(* IEC 61131-3 sources: windowtracking/test, 11 files *)

(* ---- ClearWindowTest.st ---- *)
USING AxUnit.Assert;
USING Simatic.Ax.WindowTracking.EventHandler;
USING Simatic.Ax.WindowTracking.Trigger;

NAMESPACE Simatic.Ax.WindowTracking.EventHandler
    {TestFixture}
    CLASS ClearWindowTest
        VAR PROTECTED
            tws : TransportWindowList;
            enc : EncoderMock;
            v1 : VirtualTrigger := (Position := 100, Id := UINT#1);
            v2 : VirtualTrigger := (Position := 200, Id := UINT#2);
            te1 : TriggerEventMock;
            te2 : TerminateWindowEvent;
            tl : TriggerList;
        END_VAR

        METHOD PROTECTED Setup
            tws.Encoder := enc;
            v1.EventHandler := te1;
            v2.EventHandler := te2;
            te2.WindowList := tws;
            tl.Add(v1);
            tl.Add(v2);
            tws.TriggerPointList := tl;
        END_METHOD

        {Test}
        METHOD PUBLIC Test_Clear_window
            THIS.Setup();
            tws.Create();
            enc.EncoderValue := 0;
            tws.Evaluate();
            Equal(expected := UINT#1, actual := tws.Count());

            enc.EncoderValue := 100;
            tws.Create();
            tws.Evaluate();
            Equal(expected := UINT#2, actual := tws.Count());

            // Remove Window at Position 200
            enc.EncoderValue := 200;
            tws.Evaluate();
            Equal(expected := UINT#1, actual := tws.Count());

        END_METHOD
    END_CLASS
END_NAMESPACE

(* ---- ItemTest.st ---- *)
USING AxUnit.Assert;
USING Simatic.Ax.WindowTracking.Trigger;

NAMESPACE Simatic.Ax.WindowTracking.Items
    {TestFixture}
    CLASS ItemTest
        VAR PROTECTED
            i : ItemOneDestination;
            vt : VirtualTrigger;
            ivt : IVirtualTrigger;
        END_VAR

        {Test}
        METHOD PUBLIC Test_Count_with_no_deststination_expect_0
            Equal(expected := i.DestinationCount(), actual := 0);
        END_METHOD

        {Test}
        METHOD PUBLIC Test_Count_with_1_deststination_expect_1
            i.Destination1 := vt;
            Equal(expected := i.DestinationCount(), actual := 1);
        END_METHOD

        {Test}
        METHOD PUBLIC Test_GetItem_with_no_deststination_expect_NULL
            Equal(expected := TRUE, actual := i.GetDestination() = NULL);
        END_METHOD

        {Test}
        METHOD PUBLIC Test_GetItem_with_1_deststination_expect_desztiation
            i.Destination1 := vt;
            ivt := vt;
            Equal(expected := TRUE, actual := i.GetDestination() = ivt);
        END_METHOD

    END_CLASS
END_NAMESPACE

(* ---- SortDecisionOneDestinationTest.st ---- *)
USING AxUnit.Assert;

NAMESPACE Simatic.Ax.WindowTracking
    {TestFixture}
    CLASS SortDecisionOneDestinationTest
        VAR PROTECTED
            sd : SortDecisionOneDestination;
            tw : TransportWindow;
            te : VirtualTrigger;
            te_notok : VirtualTrigger;
            ep : SortDecisionEvent;
            eph : ExitEventHandlerMock;
            item : ItemOneDestination;
        END_VAR

        METHOD PROTECTED Setup
            item.Destination1 := te;
            tw.Item := item;

            te.Id := UINT#1;
            te.Position := 1000;
            te.EventHandler := ep;

            ep.SortStrategy := sd;
            ep.ExitHandler := eph;
        END_METHOD

        {Test}
        METHOD PUBLIC Check_SortdecissonOk
            VAR_TEMP
                _check : BOOL;
            END_VAR
            THIS.Setup();
            _check := sd.Check(tw := tw, te := te, exitpoint := eph);
            Equal(expected := TRUE, actual := _check);
        END_METHOD

        {Test}
        METHOD PUBLIC Check_SortdecissonNotOk
            VAR_TEMP
                _check : BOOL;
            END_VAR
            THIS.Setup();
            _check := sd.Check(tw := tw, te := te_notok, exitpoint := eph);
            Equal(expected := FALSE, actual := _check);
        END_METHOD

    END_CLASS

    CLASS ExitEventHandlerMock IMPLEMENTS IExitPointHandler
        VAR PUBLIC

        END_VAR
        VAR PROTECTED

        END_VAR

        METHOD PUBLIC IsReady : BOOL
            IsReady := TRUE;
        END_METHOD

        METHOD PUBLIC Activate : BOOL
            ;
        END_METHOD
END_CLASS

END_NAMESPACE

(* ---- SortDecissionOneDestinationTest.st ---- *)
USING AxUnit.Assert;
USING Simatic.Ax.WindowTracking.EventHandler;
USING Simatic.Ax.WindowTracking.Trigger;
USING Simatic.Ax.WindowTracking.Items;
USING Simatic.Ax.WindowTracking.ExitPointHandler;

NAMESPACE Simatic.Ax.WindowTracking.SortDecission
    {TestFixture}
    CLASS SortDecissionOneDestinationTest
        VAR PROTECTED
            sd : SortDecissionOneDestination;
            tw : TransportWindow;
            te : VirtualTrigger;
            te_notok : VirtualTrigger;
            ep : SortDecissionEvent;
            eph : ExitEventHandlerMock;
            item : ItemOneDestination;
        END_VAR

        METHOD PROTECTED Setup
            item.Destination1 := te;
            tw.Item := item;

            te.Id := UINT#1;
            te.Position := 1000;
            te.EventHandler := ep;

            ep.SortStrategy := sd;
            ep.ExitHandler := eph;
        END_METHOD

        {Test}
        METHOD PUBLIC Check_SortdecissonOk
            VAR_TEMP
                _check : BOOL;
            END_VAR
            THIS.Setup();
            _check := sd.Check(tw := tw, te := te, exitpoint := eph);
            Equal(expected := TRUE, actual := _check);
        END_METHOD

        {Test}
        METHOD PUBLIC Check_SortdecissonNotOk
            VAR_TEMP
                _check : BOOL;
            END_VAR
            THIS.Setup();
            _check := sd.Check(tw := tw, te := te_notok, exitpoint := eph);
            Equal(expected := FALSE, actual := _check);
        END_METHOD

    END_CLASS

    CLASS ExitEventHandlerMock IMPLEMENTS IExitPointHandler
        VAR PUBLIC

        END_VAR
        VAR PROTECTED

        END_VAR

        METHOD PUBLIC IsReady : BOOL
            IsReady := TRUE;
        END_METHOD

        METHOD PUBLIC Activate : BOOL
            ;
        END_METHOD
END_CLASS

END_NAMESPACE

(* ---- TerminateWindowTest.st ---- *)
USING AxUnit.Assert;
USING Simatic.Ax.WindowTracking.EventHandler;
USING Simatic.Ax.WindowTracking.Trigger;

NAMESPACE Simatic.Ax.WindowTracking.EventHandler
    {TestFixture}
    CLASS TerminateWindowTest
        VAR PROTECTED
            tws : TransportWindowList;
            enc : EncoderMock;
            v1 : VirtualTrigger := (Position := 100, Id := UINT#1);
            v2 : VirtualTrigger := (Position := 200, Id := UINT#2);
            te1 : TriggerEventMock;
            te2 : TerminateWindowEvent;

            tl : VirtualTriggerList;
            teAfter : TerminateUserEvent;
            teBefore : TerminateUserEvent;
            TriggerPointList : ARRAY[0..50] OF IVirtualTrigger;
        END_VAR

        METHOD PROTECTED Setup
            tl.TriggerPointList := REF(TriggerPointList);
            tws.Encoder := enc;
            v1.EventHandler := te1;
            v2.EventHandler := te2;
            te2.WindowList := tws;
            tl.Add(v1);
            tl.Add(v2);
            tws.TriggerPointList := tl;

            te2.EventBefore := teBefore;
            te2.EventAfter := teAfter;
        END_METHOD

        {Test}
        METHOD PUBLIC Test_Clear_window
            THIS.Setup();
            tws.Create();
            enc.EncoderValue := 0;
            tws.Evaluate();
            Equal(expected := UINT#1, actual := tws.Count());

            enc.EncoderValue := 100;
            tws.Create();
            tws.Evaluate();
            Equal(expected := UINT#2, actual := tws.Count());

            // Remove Window at Position 200
            enc.EncoderValue := 200;
            tws.Evaluate();
            enc.EncoderValue := 206;  // move window out of range
            tws.Evaluate();
            Equal(expected := UINT#1, actual := tws.Count());

            // test for before/after event
            Equal(expected := 1, actual := teAfter.Count);
            Equal(expected := 1, actual := teBefore.Count);
        END_METHOD
    END_CLASS

    CLASS TerminateUserEvent IMPLEMENTS IUserDefinedEvent
        VAR PUBLIC
            Count : INT;
        END_VAR
        VAR PROTECTED

        END_VAR

        METHOD PUBLIC MyMethod
            ;
        END_METHOD

        METHOD PUBLIC Action : EventStatus
            VAR_INPUT
                te : IVirtualTrigger;
                tw : ITransportWindow;
            END_VAR
            Count := Count + 1;

        END_METHOD
END_CLASS
END_NAMESPACE

(* ---- test.st ---- *)
USING AxUnit;

NAMESPACE MyTest

    {TestFixture}
    CLASS MyTestFixture
        // {Test(head := 5, tail := 1, count := 4)}
        // {Test(head := 0, tail := 0, count := 1)}
        // {Test(head := 1, tail := 0, count := 1)}
        {Test(head := 0, tail := 99, count := 1)}
        METHOD PUBLIC MyTestMethod
            VAR_INPUT
                head : INT;
                tail : INT;
                count : INT;
            END_VAR
            VAR_TEMP
                result : INT;
            END_VAR
            result := (head - tail) MOD 100;
            Assert.Equal(actual := result, expected := count);
        END_METHOD
    END_CLASS

END_NAMESPACE

(* ---- TransportWindowsListTest.st ---- *)
USING AxUnit.Assert;
USING Simatic.Ax.WindowTracking.Trigger;
USING Simatic.Ax.SimpleControlModules;

NAMESPACE Simatic.Ax.WindowTracking
    {TestFixture}
    CLASS Test_WindowList

        VAR PROTECTED
            tws : TransportWindowList;
            enc : EncoderMock;
            v1 : VirtualTrigger := (Position := 100, Id := UINT#1);
            v2 : VirtualTrigger := (Position := 200, Id := UINT#2);
            te1 : TriggerEventMock;
            te2 : TriggerEventMock;
            tl : TriggerList;
        END_VAR

        METHOD PROTECTED Setup
            tws.Encoder := enc;
            v1.EventHandler := te1;
            v2.EventHandler := te2;
            tl.Add(v1);
            tl.Add(v2);
            tws.TriggerPointList := tl;
        END_METHOD

        {Test}
        METHOD PUBLIC Count_Of_Empty_List_Expect_0
            THIS.Setup();
            Equal(expected := UINT#0, actual := tws.Count());
        END_METHOD

        {Test}
        METHOD PUBLIC Remove_Window_fom_empty_list_expect_0
            THIS.Setup();
            tws.Terminate();
            Equal(expected := UINT#0, actual := tws.Count());
        END_METHOD

        {Test}
        METHOD PUBLIC Create_4Windows_And_Call_Count_Expect_4
            THIS.Setup();
            tws.Create();
            tws.Create();
            tws.Create();
            tws.Create();

            Equal(expected := UINT#4, actual := tws.Count());
        END_METHOD

        {Test}
        METHOD PUBLIC Remove_1of_4_windows_expect_count_3
            THIS.Create_4Windows_And_Call_Count_Expect_4();
            tws.Terminate();
            Equal(expected := UINT#3, actual := tws.Count());
        END_METHOD

        {Test}
        METHOD PUBLIC Remove_4of_4_windows_expect_count_0
            THIS.Create_4Windows_And_Call_Count_Expect_4();
            tws.Terminate();
            tws.Terminate();
            tws.Terminate();
            tws.Terminate();
            Equal(expected := UINT#0, actual := tws.Count());
        END_METHOD

        {Test}
        METHOD PUBLIC Remove_5of_4_windows_expect_count_0
            THIS.Create_4Windows_And_Call_Count_Expect_4();
            tws.Terminate();
            tws.Terminate();
            tws.Terminate();
            tws.Terminate();
            tws.Terminate();
            Equal(expected := UINT#0, actual := tws.Count());
        END_METHOD

        {Test}
        METHOD PUBLIC Remove_1of_4_andd_a_1_windows_expect_count_4
            THIS.Create_4Windows_And_Call_Count_Expect_4();
            tws.Terminate();
            tws.Create();
            Equal(expected := UINT#4, actual := tws.Count());
        END_METHOD

        {Test}
        METHOD PUBLIC Test_Evaluate_4_windows_with_Distance_10
            VAR_TEMP
                pos : DINT;
            END_VAR
            THIS.Create_4Windows_And_Call_Count_Expect_4();
            THIS.Setup();
            enc.EncoderValue := 10;
            tws.Evaluate();
            pos := tws.GetWindow(UINT#0).GetPosition();
            Equal(expected := 10, actual := pos);
            pos := tws.GetWindow(UINT#1).GetPosition();
            Equal(expected := 10, actual := pos);
            pos := tws.GetWindow(UINT#2).GetPosition();
            Equal(expected := 10, actual := pos);
            pos := tws.GetWindow(UINT#3).GetPosition();
            Equal(expected := 10, actual := pos);
        END_METHOD

        {Test}
        METHOD PUBLIC Test_Evaluate_4_windows_with_Distance_20
            VAR_TEMP
                pos : DINT;
            END_VAR
            THIS.Test_Evaluate_4_windows_with_Distance_10();
            enc.EncoderValue := 20;
            tws.Evaluate();
            pos := tws.GetWindow(UINT#0).GetPosition();
            Equal(expected := 20, actual := pos);
            pos := tws.GetWindow(UINT#1).GetPosition();
            Equal(expected := 20, actual := pos);
            pos := tws.GetWindow(UINT#2).GetPosition();
            Equal(expected := 20, actual := pos);
            pos := tws.GetWindow(UINT#3).GetPosition();
            Equal(expected := 20, actual := pos);
        END_METHOD

        {Test}
        METHOD PUBLIC Test_Evaluate_4_windows_with_Distance_20_remove_one_Expect_one_null
            VAR_TEMP
                pos : DINT;
                ti : ITransportWindow;
            END_VAR
            ;
            THIS.Setup();

            enc.EncoderValue := 0;
            tws.Create();
            tws.Evaluate();

            Equal(expected := UINT#1, actual := tws.Count());

            Equal(expected := te1.Id, actual := UINT#0);
            Equal(expected := te2.Id, actual := UINT#0);

            // No virtual trigger triggered
            enc.EncoderValue := 20;
            tws.Evaluate();

            Equal(expected := te1.Id, actual := UINT#0);
            Equal(expected := te2.Id, actual := UINT#0);
            Equal(expected := 0, actual := te1.Calls);
            Equal(expected := 0, actual := te2.Calls);

            // First virtual trigger triggered
            enc.EncoderValue := 99;
            tws.Evaluate();

            Equal(expected := te1.Id, actual := UINT#1);
            Equal(expected := te2.Id, actual := UINT#0);
            Equal(expected := 1, actual := te1.Calls);
            Equal(expected := 0, actual := te2.Calls);

            // First virtual trigger still occupied
            enc.EncoderValue := 100;
            tws.Evaluate();

            Equal(expected := te1.Id, actual := UINT#1);
            Equal(expected := te2.Id, actual := UINT#0);
            Equal(expected := 1, actual := te1.Calls);
            Equal(expected := 0, actual := te2.Calls);

            // Second virtual trigger still occupied
            enc.EncoderValue := 200;
            tws.Evaluate();

            Equal(expected := te1.Id, actual := UINT#1);
            Equal(expected := te2.Id, actual := UINT#2);
            Equal(expected := 1, actual := te1.Calls);
            Equal(expected := 1, actual := te2.Calls);

            // second virtual trigger triggered

            tws.Create(); // Create new window
            enc.EncoderValue := 300;
            tws.Evaluate();

            Equal(expected := te1.Id, actual := UINT#1);
            Equal(expected := te2.Id, actual := UINT#2);
            Equal(expected := 2, actual := te1.Calls);
            Equal(expected := 1, actual := te2.Calls);

            // windows moved to pos 400 - second wndow reach second trigger point
            enc.EncoderValue := 400;
            tws.Evaluate();
            Equal(expected := te1.Id, actual := UINT#1);
            Equal(expected := te2.Id, actual := UINT#2);
            Equal(expected := 2, actual := te1.Calls);
            Equal(expected := 2, actual := te2.Calls);
        END_METHOD

        {Test}
        METHOD PUBLIC Test_Null_Reference_to_Encoder
            VAR_TEMP
                tw : ITransportWindow;
            END_VAR
            tw := tws.Create();
            Equal(expected := TRUE, actual := tw = NULL);

        END_METHOD

        {Test}
        METHOD PUBLIC Create_A_window_onenocoder_value_300_and_track_the_position
            VAR_TEMP
                i : INT;
                pos : DINT;
                pos_exp : DINT;
            END_VAR
            tws.Encoder := enc;
            enc.EncoderValue := 300;
            tws.Create(); // Create new window
            FOR i := 0 TO 99 DO
                tws.Evaluate();
                pos := tws.GetWindow(UINT#0).GetPosition();
                Equal(expected := pos_exp, actual := pos);
                pos_exp := pos_exp + 100;
                enc.EncoderValue := (enc.EncoderValue + 100) MOD 4096;
            END_FOR;
            Equal(expected := 9900, actual := pos);
            ; // AxUnit.Assert.Equal(y, x)
        END_METHOD

    END_CLASS

    CLASS EncoderMock IMPLEMENTS IEncoder

        VAR PUBLIC
            EncoderValue : DINT;
        END_VAR

        METHOD PUBLIC Evaluate
            ;
        END_METHOD

        METHOD PUBLIC Reset
            ;
        END_METHOD

        METHOD PUBLIC SetValue
            VAR_INPUT
                value : DINT;
            END_VAR
            ;
        END_METHOD

        METHOD PUBLIC GetValue : DINT
            GetValue := EncoderValue;
        END_METHOD

        METHOD PUBLIC SetDirection
            VAR_INPUT
                mode : CountMode;
            END_VAR
            ;
        END_METHOD

        METHOD PUBLIC RelativeCount : DINT
            ;
        END_METHOD

        METHOD PUBLIC ResetRelative
            ;
        END_METHOD

        METHOD PUBLIC GetModulo : DINT
            GetModulo := 4096;
        END_METHOD
    END_CLASS

END_NAMESPACE

(* ---- TransportWindowTest.st ---- *)
USING AxUnit.Assert;
USING Simatic.Ax.WindowTracking.Trigger;
USING Simatic.Ax.SimpleControlModules;

NAMESPACE Simatic.Ax.WindowTracking
    {TestFixture}
    CLASS Test_TransportWindowList

        VAR PROTECTED
            tw : TransportWindow;
            enc : EncoderMock;
        END_VAR

        {Test}
        METHOD PUBLIC CalcPosition_of_different_encoder_values_with_offset
            tw.SetPosition(100);
            enc.EncoderValue := 0;
            tw.CalcPosition(enc);
            Equal(expected := 100, actual := tw.GetPosition());

            enc.EncoderValue := 10;
            tw.CalcPosition(enc);
            Equal(expected := 110, actual := tw.GetPosition());

            enc.EncoderValue := 4095;
            tw.CalcPosition(enc);
            Equal(expected := 4195, actual := tw.GetPosition());

            enc.EncoderValue := 1;
            tw.CalcPosition(enc);
            Equal(expected := 4197, actual := tw.GetPosition());

        END_METHOD

        {Test}
        METHOD PUBLIC CalcPosition_of_different_encoder_positions_starting_with_0
            enc.EncoderValue := 0;
            tw.CalcPosition(enc);
            Equal(expected := 0, actual := tw.GetPosition());

            enc.EncoderValue := 10;
            tw.CalcPosition(enc);
            Equal(expected := 10, actual := tw.GetPosition());

            enc.EncoderValue := 4095;
            tw.CalcPosition(enc);
            Equal(expected := 4095, actual := tw.GetPosition());

            enc.EncoderValue := 1;
            tw.CalcPosition(enc);
            Equal(expected := 4097, actual := tw.GetPosition());

        END_METHOD

        {Test}
        METHOD PUBLIC CalcPosition_of_different_encoder_positions_starting_with_100
            enc.EncoderValue := 100;
            tw.CalcPosition(enc);
            Equal(expected := 0, actual := tw.GetPosition());

            enc.EncoderValue := 110;
            tw.CalcPosition(enc);
            Equal(expected := 10, actual := tw.GetPosition());

            enc.EncoderValue := 4095;
            tw.CalcPosition(enc);
            Equal(expected := 3995, actual := tw.GetPosition());

            enc.EncoderValue := 1;
            tw.CalcPosition(enc);
            Equal(expected := 3997, actual := tw.GetPosition());

        END_METHOD

    END_CLASS

END_NAMESPACE

(* ---- VirtualTriggerListTest.st ---- *)
USING Simatic.Ax.WindowTracking.Trigger;
USING AxUnit.Assert;
NAMESPACE Simatic.Ax.WindowTracking.Trigger
    {TestFixture}
    CLASS TestVirtualTriggerList
        VAR PROTECTED
            tl : VirtualTriggerList;
            TriggerPointList : ARRAY[0..50] OF IVirtualTrigger;
            trig1 : VirtualTrigger := (Id := UINT#1, Position := 1100);
            trig2 : VirtualTrigger := (Id := UINT#2, Position := 1200);
            trig3 : VirtualTrigger := (Id := UINT#3, Position := 1300);
            trig4 : VirtualTrigger := (Id := UINT#4, Position := 1400);
            evt : TriggerEventMock;
        END_VAR

        METHOD PRIVATE SetupTriggerList
            tl.TriggerPointList := REF(TriggerPointList);
            trig1.EventHandler := evt;
            tl.Add(tp := trig1);

            trig2.EventHandler := evt;
            tl.Add(tp := trig2);

            trig3.EventHandler := evt;
            tl.Add(tp := trig3);

            trig4.EventHandler := evt;
            tl.Add(tp := trig4);
        END_METHOD

        {Test}
        METHOD PUBLIC TestCount_elements_expect_4
            THIS.SetupTriggerList();
            Equal(expected := UINT#4, actual := tl.Count());
        END_METHOD

        {Test}
        METHOD PUBLIC Test_GetId_element_not_found_expect_null
            VAR_TEMP
                t : IVirtualTrigger;
            END_VAR
            tl.TriggerPointList := REF(TriggerPointList);
            t := tl.GetTriggerPoint(UINT#1);
            Equal(expected := TRUE, actual := t = NULL);
        END_METHOD

        {Test(id := UINT#1, expVal := 1100)}
        {Test(id := UINT#2, expVal := 1200)}
        {Test(id := UINT#3, expVal := 1300)}
        {Test(id := UINT#4, expVal := 1400)}
        METHOD PUBLIC Test_GetId_of_four_triggers_and_expect_correct_position
            VAR_INPUT
                id : UINT;
                expVal : DINT;
            END_VAR
            VAR_TEMP
                vt : IVirtualTrigger;
                pos : DINT;
            END_VAR
            THIS.SetupTriggerList();
            vt := tl.GetTriggerPoint(id);
            pos := vt.GetPosition();
            Equal(expected := expVal, actual := tl.GetTriggerPoint(id).GetPosition());
        END_METHOD

    END_CLASS

    CLASS VirtualTriggerMock
        VAR PUBLIC

        END_VAR
        VAR PROTECTED

        END_VAR

        METHOD PUBLIC MyMethod
            ;
        END_METHOD
    END_CLASS

END_NAMESPACE

(* ---- VirtualTriggerTest.st ---- *)
USING AxUnit.Assert;
USING Simatic.Ax.WindowTracking.Trigger;
USING Simatic.Ax.WindowTracking.EventHandler;
NAMESPACE Simatic.Ax.WindowTracking.Trigger
    {TestFixture}
    CLASS TestVirtualTrigger
        VAR PROTECTED
            vt : VirtualTrigger;
            evt : TriggerEventMock;
            tw : TransportWindow;
            enc : EncoderMock;
        END_VAR

        METHOD PRIVATE SetupTestTrigger
            vt.EventHandler := evt;
            vt.Position := 1000;
            vt.Id := UINT#10;
        END_METHOD

        {Test}
        METHOD PUBLIC Test_Activate_method_with_no_event_expect_NullReferecne
            VAR_TEMP
                s : EventStatus;
                i : Int;
            END_VAR
            Equal(expected := TRUE, actual := s <> EventStatus#Finished);
            s := vt.ActivateEvent();
            Equal(expected := TRUE, actual := s = EventStatus#NullReference);
        END_METHOD

        {Test}
        METHOD PUBLIC Test_Activate_method_end_check_Execution
            VAR_TEMP
                s : EventStatus;
                i : Int;
            END_VAR
            THIS.SetupTestTrigger();
            Equal(expected := TRUE, actual := s <> EventStatus#Finished);
            s := vt.ActivateEvent();
            Equal(expected := TRUE, actual := s = EventStatus#Finished);
        END_METHOD

        {Test}
        METHOD PUBLIC Test_GetId_And_Expect_10
            THIS.SetupTestTrigger();
            Equal(expected := UINT#10, actual := vt.GetId());
        END_METHOD
        {Test}

        METHOD PUBLIC Test_GetPosition_And_Expect_1000
            THIS.SetupTestTrigger();
            Equal(expected := UINT#1000, actual := vt.GetPosition());
        END_METHOD

        METHOD PUBLIC Test_IsEnabled_And_Exect_true
            THIS.SetupTestTrigger();
            Equal(expected := TRUE, actual := vt.IsEnabled());
        END_METHOD

        {Test(sp := -6, res := FALSE)}
        {Test(sp := -5, res := TRUE)}
        {Test(sp := -4, res := TRUE)}
        {Test(sp := -1, res := TRUE)}
        {Test(sp := 0, res := TRUE)}
        {Test(sp := 1, res := TRUE)}
        {Test(sp := 4, res := TRUE)}
        {Test(sp := 5, res := TRUE)}
        {Test(sp := 6, res := FALSE)}
        METHOD PUBLIC Test_Check
            VAR_INPUT
                sp : DINT;
                res : BOOL;
            END_VAR
            VAR_TEMP
                r : BOOL;
            END_VAR

            vt.Position := sp;
            r := vt.Check(tw := tw, ul := 5, ll := 5);
            Equal(expected := res, actual := r);
            Equal(expected := res, actual := vt.IsActivated());

            r := vt.Check(tw := tw, ul := 5, ll := 5);
            Equal(expected := FALSE, actual := r);
            Equal(expected := res, actual := vt.IsActivated());
        END_METHOD

        {Test}
        METHOD PUBLIC TestCheckforRisingEdge_expect_just_one_rising_edge

            vt.Position := 100;

            enc.EncoderValue := 0;
            tw.CalcPosition(enc := enc);
            Equal(expected := 0, actual := tw.GetPosition());
            Equal(expected := FALSE, actual := vt.Check(tw := tw, ul := 5, ll := 5));

            enc.EncoderValue := 1;
            tw.CalcPosition(enc := enc);
            Equal(expected := 1, actual := tw.GetPosition());
            Equal(expected := FALSE, actual := vt.Check(tw := tw, ul := 5, ll := 5));

            enc.EncoderValue := 94;
            tw.CalcPosition(enc := enc);
            Equal(expected := 94, actual := tw.GetPosition());
            Equal(expected := FALSE, actual := vt.Check(tw := tw, ul := 5, ll := 5));

            enc.EncoderValue := 95;
            tw.CalcPosition(enc := enc);
            Equal(expected := 95, actual := tw.GetPosition());
            Equal(expected := TRUE, actual := vt.Check(tw := tw, ul := 5, ll := 5));

            enc.EncoderValue := 96;
            tw.CalcPosition(enc := enc);
            Equal(expected := 96, actual := tw.GetPosition());
            Equal(expected := FALSE, actual := vt.Check(tw := tw, ul := 5, ll := 5));

            enc.EncoderValue := 97;
            tw.CalcPosition(enc := enc);
            Equal(expected := 97, actual := tw.GetPosition());
            Equal(expected := FALSE, actual := vt.Check(tw := tw, ul := 5, ll := 5));

            enc.EncoderValue := 98;
            tw.CalcPosition(enc := enc);
            Equal(expected := 98, actual := tw.GetPosition());
            Equal(expected := FALSE, actual := vt.Check(tw := tw, ul := 5, ll := 5));

            enc.EncoderValue := 105;
            tw.CalcPosition(enc := enc);
            Equal(expected := 105, actual := tw.GetPosition());
            Equal(expected := FALSE, actual := vt.Check(tw := tw, ul := 5, ll := 5));

            enc.EncoderValue := 194;
            tw.CalcPosition(enc := enc);
            Equal(expected := 194, actual := tw.GetPosition());
            Equal(expected := FALSE, actual := vt.Check(tw := tw, ul := 5, ll := 5));

            tw.Reset();
            enc.EncoderValue := 194;
            tw.CalcPosition(enc := enc);
            Equal(expected := 0, actual := tw.GetPosition());
            Equal(expected := FALSE, actual := vt.Check(tw := tw, ul := 5, ll := 5));

            enc.EncoderValue := 288;
            tw.CalcPosition(enc := enc);
            Equal(expected := 94, actual := tw.GetPosition());
            Equal(expected := FALSE, actual := vt.Check(tw := tw, ul := 5, ll := 5));

            enc.EncoderValue := 289;
            tw.CalcPosition(enc := enc);
            Equal(expected := 95, actual := tw.GetPosition());
            Equal(expected := TRUE, actual := vt.Check(tw := tw, ul := 5, ll := 5));

        END_METHOD

    END_CLASS

    CLASS TriggerEventMock IMPLEMENTS ITriggerEvent
        VAR PUBLIC
            Id : UINT;
            Calls : INT;
        END_VAR
        VAR PROTECTED

        END_VAR

        METHOD PUBLIC Action : EventStatus
            VAR_INPUT
                te : IVirtualTrigger;
                tw : ITransportWindow;
            END_VAR

            Id := te.GetId();
            Action := EventStatus#Finished;
            Calls := Calls + 1;
        END_METHOD

    END_CLASS
END_NAMESPACE

(* ---- WindowingIntegrativeTest.st ---- *)
USING AxUnit.Assert;
USING Simatic.Ax.WindowTracking.Trigger;
USING Simatic.Ax.WindowTracking.EventHandler;
NAMESPACE Simatic.Ax.WindowTracking.Trigger
    {TestFixture}
    CLASS WindowingIntegraiveTest
        VAR PROTECTED
            twl : TransportWindowList;
            tpl : VirtualTriggerList;

            tp1 : VirtualTrigger;
            hdl : EventHandlerTest;
            tw : TransportWindow;
            enc : EncoderMock;
        END_VAR

        METHOD PUBLIC Setup
            twl.Encoder := enc;
            twl.TriggerPointList := tpl;

            tp1.Position := 100;
            tp1.Id := UINT#1;
            tp1.EventHandler := hdl;
            tpl.Add(tp1);
        END_METHOD

        {Test}
        METHOD PUBLIC Test_Crate3_Windows_with_distance_20
            THIS.Setup();
            // Position 0 Create window
            enc.EncoderValue := 0;
            twl.Create();
            twl.Evaluate();
            Equal(expected := 0, actual := twl.GetWindow(UINT#0).GetPosition());

            // Position 20 Create 2. window
            enc.EncoderValue := 20;
            twl.Create();
            twl.Evaluate();
            Equal(expected := 20, actual := twl.GetWindow(UINT#0).GetPosition());
            Equal(expected := 0, actual := twl.GetWindow(UINT#1).GetPosition());

            // Position 40 Create 3. window
            enc.EncoderValue := 40;
            twl.Create();
            twl.Evaluate();
            Equal(expected := 40, actual := twl.GetWindow(UINT#0).GetPosition());
            Equal(expected := 20, actual := twl.GetWindow(UINT#1).GetPosition());
            Equal(expected := 0, actual := twl.GetWindow(UINT#2).GetPosition());

        END_METHOD

        {Test}
        METHOD PUBLIC Move_First_window_to_triggerpoint_at_position_95_and_expect_activation
            THIS.Test_Crate3_Windows_with_distance_20();
            enc.EncoderValue := 94;
            twl.Evaluate();
            Equal(expected := 94, actual := twl.GetWindow(UINT#0).GetPosition());
            Equal(expected := 74, actual := twl.GetWindow(UINT#1).GetPosition());
            Equal(expected := 54, actual := twl.GetWindow(UINT#2).GetPosition());

            Equal(expected := FALSE, actual :=  tp1.IsActivated());

            enc.EncoderValue := 95;
            twl.Evaluate();
            Equal(expected := TRUE, actual :=  tp1.IsActivated());
            Equal(expected := 1, actual := hdl.Count);

            enc.EncoderValue := 96;
            twl.Evaluate();
            Equal(expected := TRUE, actual :=  tp1.IsActivated());
            Equal(expected := 1, actual := hdl.Count);

            enc.EncoderValue := 105;
            twl.Evaluate();
            Equal(expected := TRUE, actual :=  tp1.IsActivated());
            Equal(expected := 1, actual := hdl.Count);

            enc.EncoderValue := 106;
            twl.Evaluate();
            Equal(expected := TRUE, actual :=  tp1.IsActivated());
            Equal(expected := 1, actual := hdl.Count);
        END_METHOD

    END_CLASS

    CLASS EventHandlerTest IMPLEMENTS ITriggerEvent
        VAR PUBLIC
            Count : DINT;
        END_VAR

        METHOD PUBLIC Action : EventStatus
            VAR_INPUT
                te : IVirtualTrigger;
                tw : ITransportWindow;
            END_VAR
            Count := Count + 1;
        END_METHOD
    END_CLASS

END_NAMESPACE
